# EPICS autosave request: iocBoot/iocKetek/auto_settings.req
file "ketek_settings.req",        P=$(P), R=$(R)
file "mca_settings.req",          P=$(P), M=$(M)
#file "commonPlugin_settings.req", P=$(P)
